// TIA Portal V15.1 export
// export: Created 2020-06-12T07:35:48.8037109Z, ExportSetting None, DisplayName Totally Integrated Automation Portal, DisplayVersion V15.1, DisplayName TIA Portal Openness, DisplayVersion V15.1, DisplayName STEP 7 Professional, DisplayVersion V15.1, DisplayName STEP 7 Safety, DisplayVersion V15.1, DisplayName WinCC Advanced, DisplayVersion V15.1
FUNCTION "PWR_meas" : Void   // FC148, FBD
{ S7_Optimized_Access := 'TRUE' }
// stored: SetENOAutomatically False
   VAR_TEMP
      tFiltLen : Int;
   END_VAR
   VAR_TEMP   // added for the SCL form of the ladder/FBD networks
      _w1 : Bool;
   END_VAR
BEGIN

REGION Network 1: Actual Current, kA
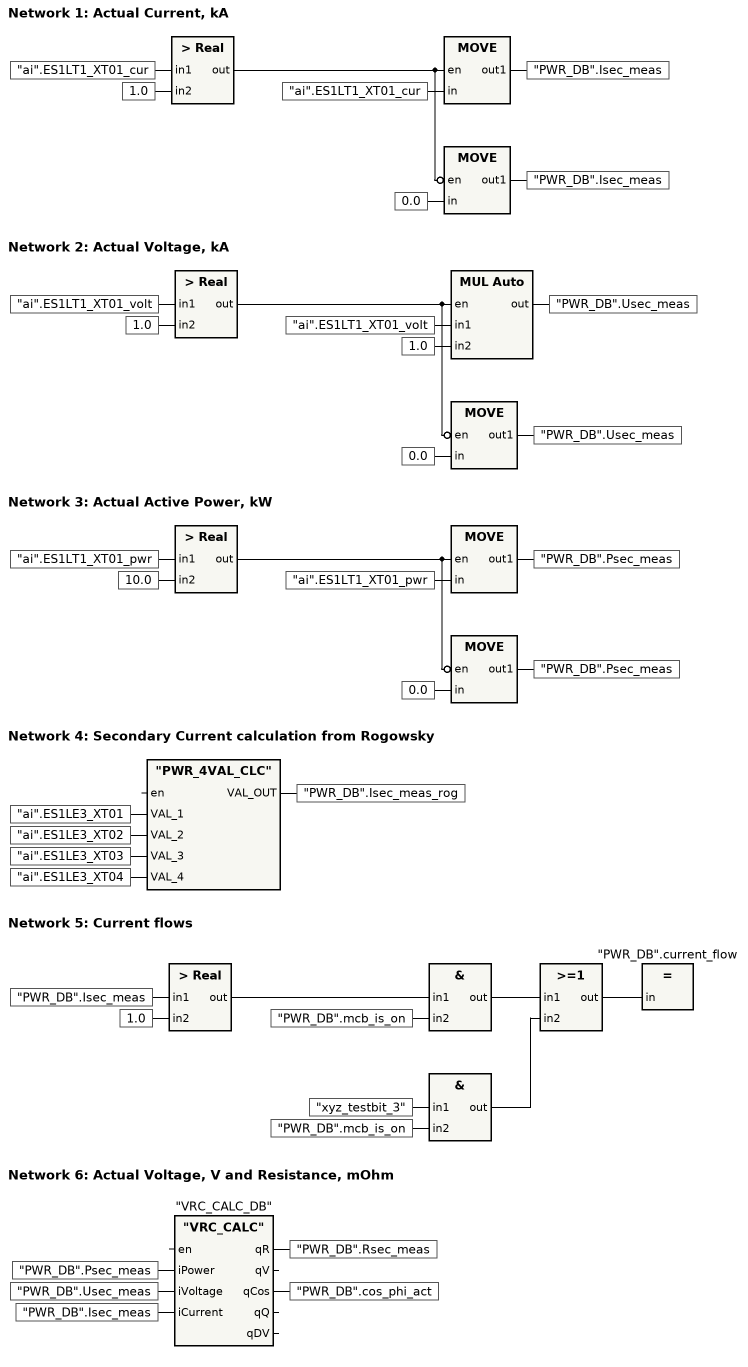
   #_w1 := "ai".ES1LT1_XT01_cur > 1.0;
   IF #_w1 THEN "PWR_DB".Isec_meas := "ai".ES1LT1_XT01_cur; END_IF;
   IF NOT #_w1 THEN "PWR_DB".Isec_meas := 0.0; END_IF;
END_REGION

REGION Network 2: Actual Voltage, kA
   // I use factor beacuse the measurement line has gain which is not equal 1
   // K = 1.12167
   // PuM/2019-05-29 : I connect Sineax M563 directly to the transformer. K = 1
   #_w1 := "ai".ES1LT1_XT01_volt > 1.0;
   IF #_w1 THEN "PWR_DB".Usec_meas := "ai".ES1LT1_XT01_volt * 1.0; END_IF;
   IF NOT #_w1 THEN "PWR_DB".Usec_meas := 0.0; END_IF;
END_REGION

REGION Network 3: Actual Active Power, kW
   #_w1 := "ai".ES1LT1_XT01_pwr > 10.0;
   IF #_w1 THEN "PWR_DB".Psec_meas := "ai".ES1LT1_XT01_pwr; END_IF;
   IF NOT #_w1 THEN "PWR_DB".Psec_meas := 0.0; END_IF;
END_REGION

REGION Network 4: Secondary Current calculation from Rogowsky
   "PWR_4VAL_CLC"(VAL_1 := "ai".ES1LE3_XT01,
                  VAL_2 := "ai".ES1LE3_XT02,
                  VAL_3 := "ai".ES1LE3_XT03,
                  VAL_4 := "ai".ES1LE3_XT04,
                  VAL_OUT => "PWR_DB".Isec_meas_rog);
END_REGION

REGION Network 5: Current flows
   "PWR_DB".current_flow := (("PWR_DB".Isec_meas > 1.0) AND "PWR_DB".mcb_is_on) OR ("xyz_testbit_3" AND "PWR_DB".mcb_is_on);
END_REGION

REGION Network 6: Actual Voltage, V and Resistance, mOhm
   "VRC_CALC_DB"(iPower := "PWR_DB".Psec_meas,   // "VRC_CALC"
                 iVoltage := "PWR_DB".Usec_meas,
                 iCurrent := "PWR_DB".Isec_meas,
                 qR => "PWR_DB".Rsec_meas,
                 qCos => "PWR_DB".cos_phi_act);
END_REGION

REGION Network 7: Cos(phi) filtration
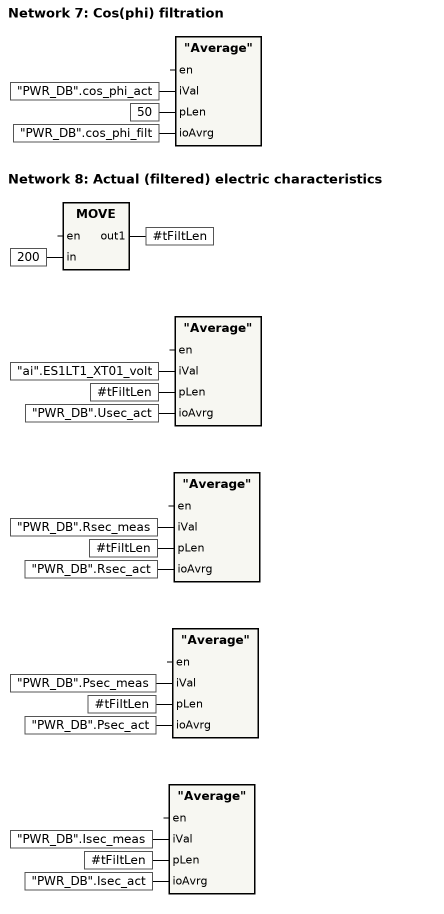
   "Average"(iVal := "PWR_DB".cos_phi_act, pLen := 50, ioAvrg := "PWR_DB".cos_phi_filt);
END_REGION

REGION Network 8: Actual (filtered) electric characteristics
   #tFiltLen := 200;
   "Average"(iVal := "ai".ES1LT1_XT01_volt, pLen := #tFiltLen, ioAvrg := "PWR_DB".Usec_act);
   "Average"(iVal := "PWR_DB".Rsec_meas, pLen := #tFiltLen, ioAvrg := "PWR_DB".Rsec_act);
   "Average"(iVal := "PWR_DB".Psec_meas, pLen := #tFiltLen, ioAvrg := "PWR_DB".Psec_act);
   "Average"(iVal := "PWR_DB".Isec_meas, pLen := #tFiltLen, ioAvrg := "PWR_DB".Isec_act);
END_REGION
END_FUNCTION
